{attribute addProperty BoxType "EK1100-0000-0018"}
{attribute addProperty Id "Beckhoff_EJ5xxxEK1122Beckhoff_EJ5xxxEK1122_0744EC7C162A_0001_EJ5002_0000_0016EJ5002_8CF434FD19224A_0002_EJ5002_0000_0017EJ5002_D767A13319224A_0003_EJ5101_0000_0016EJ5101_AD0B958A17622A_0004_EJ5151_0000_0016EJ5151_3376D36320826"}
{attribute addProperty CRC "2422587745"}
{attribute addProperty SizeInBites "784"}
{attribute addProperty SizeInBytes "98"}
TYPE Beckhoff_EJ5xxx_9065C161 EXTENDS EK1100_179A0949 :
STRUCT
	{attribute addProperty Name "Beckhoff_EJ5xxxEK1122"}
	Beckhoff_EJ5xxxEK1122 : Beckhoff_EJ5xxxEK1122_0744EC7C;
	{attribute addProperty Name "A_0001_EJ5002_0000_0016"}
	A_0001_EJ5002_0000_0016 : EJ5002_8CF434FD;
	{attribute addProperty Name "A_0002_EJ5002_0000_0017"}
	A_0002_EJ5002_0000_0017 : EJ5002_D767A133;
	{attribute addProperty Name "A_0003_EJ5101_0000_0016"}
	A_0003_EJ5101_0000_0016 : EJ5101_AD0B958A;
	{attribute addProperty Name "A_0004_EJ5151_0000_0016"}
	A_0004_EJ5151_0000_0016 : EJ5151_3376D363;
END_STRUCT
END_TYPE

(* stored: Version 1.2.0.0, ProductVersion 3.1.4024.9
   DUT Beckhoff_EJ5xxx_9065C161: Id {274ec41b-6bad-4cbc-b6ac-55a4d26e9aa9} *)
